/// Declaration of a distinct unit of this application
FUNCTION_BLOCK HandlingUnit EXTENDS ZApplication.Unit IMPLEMENTS IHandling
VAR
  _equipment : HandlingEquipment(THIS^);
  _data : HandlingDataRef;
  _com : HandlingComRef;

  _boot : HandlingSequenceBoot(THIS^);
  _automatic : HandlingSequenceAutomatic(THIS^);
  _stop : HandlingSequenceStop(THIS^);
  _gohome : HandlingSequenceGoHome(THIS^);
  _faultReaction : HandlingSequenceFaultReaction(THIS^);
  
  _statemachine : ZApplication.UnitStateMachine;

  _observeTimer : ZAux.Timer;
END_VAR

{attribute 'ZId' := '2160a0d9-b961-4504-830a-bd7771ead3e7'}

IF _observeTimer.Done THEN
  _observeTimer.WaitAsync(0.1);
  
  // monitor _com for requested actions (e.g. start homing, start automatic mode, ...)
  ObserveRequest(_com.Subscribe.Request.Start, ZApplication.UnitStateMachineState.Automatic);
  ObserveRequest(_com.Subscribe.Request.Stop, ZApplication.UnitStateMachineState.Stop);
  ObserveRequest(_com.Subscribe.Request.GoHome, ZApplication.UnitStateMachineState.GoHome);
  ObserveRequest(_com.Subscribe.Request.Halt, ZApplication.UnitStateMachineState.Halt);
  
  // provide relevant information via ADS
  _com.Publish.Request.Stop := _stateMachine.IsTransitionAllowed(ZApplication.UnitStateMachineState.Stop);
  _com.Publish.Request.Start := _stateMachine.IsTransitionAllowed(ZApplication.UnitStateMachineState.Automatic);
  _com.Publish.Request.GoHome := _stateMachine.IsTransitionAllowed(ZApplication.UnitStateMachineState.GoHome);
  _com.Publish.Request.Halt := _stateMachine.IsTransitionAllowed(ZApplication.UnitStateMachineState.Halt);

  _com.Publish.State := _stateMachine.State();
END_IF

IF _statemachine.State() <> UnitStateMachineState.Automatic
THEN
  _equipment.Collision.Joint1.SetPosition((_equipment.Axis.Axis1.ActualPosition + _equipment.Axis.Axis1.ActualFollowingError) / 180.0 * ZCore.Constants.Pi);
  _equipment.Collision.Joint2.SetPosition((_equipment.Axis.Axis2.ActualPosition + _equipment.Axis.Axis2.ActualFollowingError) / 180.0 * ZCore.Constants.Pi);
  _equipment.Collision.Joint3.SetPosition((_equipment.Axis.Axis3.ActualPosition + _equipment.Axis.Axis3.ActualFollowingError) / 180.0 * ZCore.Constants.Pi);
END_IF

METHOD FB_init : BOOL
VAR_INPUT
  bInitRetains : BOOL; // if TRUE, the retain variables are initialized (warm start / cold start)
  bInCopyCode : BOOL;  // if TRUE, the instance afterwards gets moved into the copy code (online change)
  parent : ZCore.IManagedObject; // caller of the Unit's cyclic method. If the Unit runs in its own context use 0
  displayName : ZCore.ZString;  // name of this unit as it should show up in the logger
  configdata : REFERENCE TO HandlingDataConfig;  // reference to the configuration data that is used during boot to configure the Units equipment
  machinedata : REFERENCE TO HandlingDataMachine; // reference to the machine data that is used through most sequences of the unit (motor speed, axes positions, ...)
  calibrationdata : REFERENCE TO HandlingDataCalibration;  // reference to calibration that is determined by calibration sequences of the unit (static offsets, shifts)
  com : REFERENCE TO HandlingCom;  // reference to the communication interface that is used to control this Unit via ADS
END_VAR
_name := displayName;

// initialize local logger decorator
_loggerDecorator.FB_init(bInitRetains, bInCopyCode, _name, ZModuleProgram.Logger);
_alarmingDecorator.FB_init(bInitRetains, bInCopyCode, _name, ZModuleProgram.Alarming);

// setup data
_data.Config REF= configdata;
_data.Machine REF= machinedata;
_data.Calibration REF= calibrationdata;
_com.Publish REF= com.Publish;
_com.Subscribe REF= com.Subscribe;

// ------- sequence initialization, map sequences of this unit to the statemachine -------
{attribute '__ZwPlcUnitInitSequenceImplementation__'} // Do not remove this attribute! It is used for code generation.
_statemachine.SetSequence(ZApplication.UnitStateMachineState.Boot, _boot);
_statemachine.SetSequence(ZApplication.UnitStateMachineState.FaultReaction, _faultReaction);
_statemachine.SetSequence(ZApplication.UnitStateMachineState.Gohome, _gohome);
_statemachine.SetSequence(ZApplication.UnitStateMachineState.Stop, _stop);
_statemachine.SetSequence(ZApplication.UnitStateMachineState.Automatic, _automatic);

_statemachine.SetName(_name);
_statemachine.SetLogger(_logger);

// set initial state
_statemachine.SetState(ZApplication.UnitStateMachineState.Boot);
SetStateMachine(_statemachine);
END_METHOD

END_FUNCTION_BLOCK

(* stored: Version 1.1.0.1
   POU HandlingUnit: Id {5e765d90-464d-45c9-8a2b-1bdfc1828c8e}, SpecialFunc None
   Folder UnitInterface: Id {a0ebf69d-b69a-49ae-acc3-2a1f8aa4e0ea}
   Method FB_init: Id {a96b64eb-d71e-4687-a544-68ab74efc324} *)
